{attribute addProperty BoxType "BK1250-0000-0019"}
{attribute addProperty Id "Term_388_KL1002KL1002_D229A9CA00"}
{attribute addProperty CRC "1537847932"}
{attribute addProperty SizeInBites "0"}
{attribute addProperty SizeInBytes "0"}
TYPE A_0018_BK1250_0000_0019_5BA9B27C EXTENDS BK1250_4487A81F :
STRUCT
	{attribute addProperty Name "Term_388_KL1002"}
	Term_388_KL1002 : KL1002_D229A9CA;
END_STRUCT
END_TYPE

(* stored: Version 1.2.0.0, ProductVersion 3.1.4024.9
   DUT A_0018_BK1250_0000_0019_5BA9B27C: Id {7f669f85-b67b-43ab-a0bb-070c8dff8cdc} *)
